// TIA Portal V20 export
FUNCTION_BLOCK "Simulation"   // FB32840, LAD
// stored: MemoryReserve 100, Namespace Unit1.Em8, SetENOAutomatically false
   VAR_INPUT
      simulation { ExternalAccessible := 'False'; ExternalVisible := 'False'; ExternalWritable := 'False'} : Bool;
   END_VAR
   VAR
      instActuator { ExternalAccessible := 'False'; ExternalVisible := 'False'; ExternalWritable := 'False'} : Array[0..9] of "Simulation_Actuator";
      statDigitalSignal { ExternalAccessible := 'False'; ExternalVisible := 'False'; ExternalWritable := 'False'} : Array[0..9] of Bool;
   END_VAR
   VAR_TEMP   // added for the SCL form of the ladder/FBD networks
      _w1 : Bool;
      _w2 : Bool;
      _w3 : Bool;
   END_VAR
BEGIN

REGION Network 1: Digital Signal
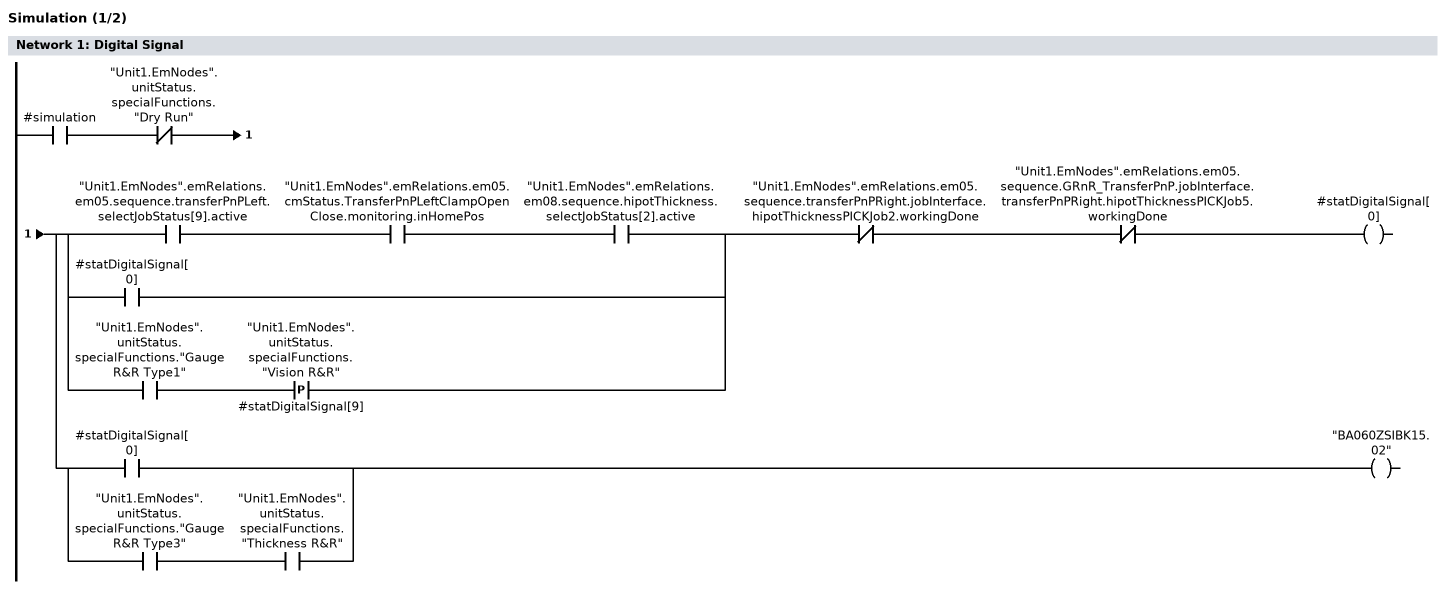
   RUNG wire#powerrail
      Contact( #simulation )
      I_Contact( "Unit1.EmNodes".unitStatus.specialFunctions."Dry Run" )
      wire#w1
      Contact( "Unit1.EmNodes".emRelations.em05.sequence.transferPnPLeft.selectJobStatus[9].active )
      Contact( "Unit1.EmNodes".emRelations.em05.cmStatus.TransferPnPLeftClampOpenClose.monitoring.inHomePos )
      Contact( "Unit1.EmNodes".emRelations.em08.sequence.hipotThickness.selectJobStatus[2].active )
      wire#w2
      I_Contact( "Unit1.EmNodes".emRelations.em05.sequence.transferPnPRight.jobInterface.hipotThicknessPICKJob2.workingDone )
      I_Contact( "Unit1.EmNodes".emRelations.em05.sequence.GRnR_TransferPnP.jobInterface.transferPnPRight.hipotThicknessPICKJob5.workingDone )
      Coil( #statDigitalSignal[0] )
   END_RUNG
   RUNG wire#w1
      Contact( #statDigitalSignal[0] )
   END_RUNG wire#w2
   RUNG wire#w1
      Contact( "Unit1.EmNodes".unitStatus.specialFunctions."Gauge R&R Type1" )
      P_Contact(operand := "Unit1.EmNodes".unitStatus.specialFunctions."Vision R&R", bit := #statDigitalSignal[9])
   END_RUNG wire#w2
   RUNG wire#w1
      Contact( #statDigitalSignal[0] )
      wire#w3
      Coil( "BA060ZSIBK15.02" )
   END_RUNG
   RUNG wire#w1
      Contact( "Unit1.EmNodes".unitStatus.specialFunctions."Gauge R&R Type3" )
      Contact( "Unit1.EmNodes".unitStatus.specialFunctions."Thickness R&R" )
   END_RUNG wire#w3
   // the same network as SCL:
   #_w1 := #simulation AND NOT "Unit1.EmNodes".unitStatus.specialFunctions."Dry Run";
   #_w3 := #_w1 AND #statDigitalSignal[0];
   #_w2 := #_w1 AND "Unit1.EmNodes".unitStatus.specialFunctions."Gauge R&R Type1" AND "Unit1.EmNodes".unitStatus.specialFunctions."Vision R&R" AND NOT #statDigitalSignal[9];   // rising edge of "Unit1.EmNodes".unitStatus.specialFunctions."Vision R&R"
   #statDigitalSignal[9] := "Unit1.EmNodes".unitStatus.specialFunctions."Vision R&R";
   #statDigitalSignal[0] := ((#_w1 AND "Unit1.EmNodes".emRelations.em05.sequence.transferPnPLeft.selectJobStatus[9].active AND "Unit1.EmNodes".emRelations.em05.cmStatus.TransferPnPLeftClampOpenClose.monitoring.inHomePos AND "Unit1.EmNodes".emRelations.em08.sequence.hipotThickness.selectJobStatus[2].active) OR #_w3 OR #_w2) AND NOT "Unit1.EmNodes".emRelations.em05.sequence.transferPnPRight.jobInterface.hipotThicknessPICKJob2.workingDone AND NOT "Unit1.EmNodes".emRelations.em05.sequence.GRnR_TransferPnP.jobInterface.transferPnPRight.hipotThicknessPICKJob5.workingDone;
   "BA060ZSIBK15.02" := #_w1 AND (#statDigitalSignal[0] OR ("Unit1.EmNodes".unitStatus.specialFunctions."Gauge R&R Type3" AND "Unit1.EmNodes".unitStatus.specialFunctions."Thickness R&R"));
END_REGION

REGION Network 2: Two Way Actuator
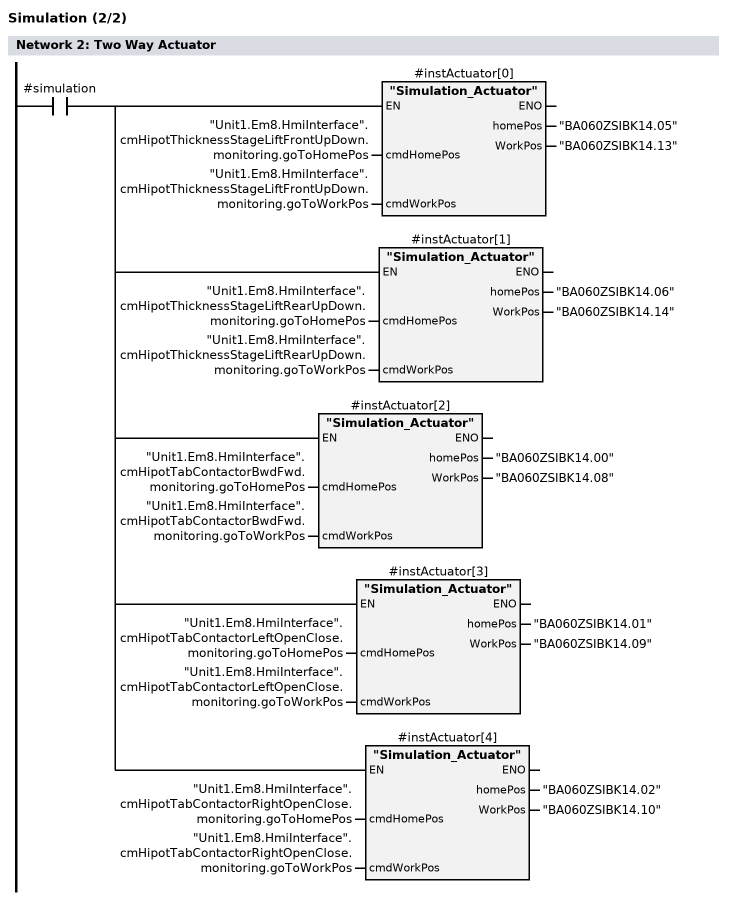
   RUNG wire#powerrail
      Contact( #simulation )
      wire#w1
      #instActuator[0](cmdHomePos := "Unit1.Em8.HmiInterface".cmHipotThicknessStageLiftFrontUpDown.monitoring.goToHomePos, cmdWorkPos := "Unit1.Em8.HmiInterface".cmHipotThicknessStageLiftFrontUpDown.monitoring.goToWorkPos, homePos => "BA060ZSIBK14.05", WorkPos => "BA060ZSIBK14.13")
   END_RUNG
   RUNG wire#w1
      #instActuator[1](cmdHomePos := "Unit1.Em8.HmiInterface".cmHipotThicknessStageLiftRearUpDown.monitoring.goToHomePos, cmdWorkPos := "Unit1.Em8.HmiInterface".cmHipotThicknessStageLiftRearUpDown.monitoring.goToWorkPos, homePos => "BA060ZSIBK14.06", WorkPos => "BA060ZSIBK14.14")
   END_RUNG
   RUNG wire#w1
      #instActuator[2](cmdHomePos := "Unit1.Em8.HmiInterface".cmHipotTabContactorBwdFwd.monitoring.goToHomePos, cmdWorkPos := "Unit1.Em8.HmiInterface".cmHipotTabContactorBwdFwd.monitoring.goToWorkPos, homePos => "BA060ZSIBK14.00", WorkPos => "BA060ZSIBK14.08")
   END_RUNG
   RUNG wire#w1
      #instActuator[3](cmdHomePos := "Unit1.Em8.HmiInterface".cmHipotTabContactorLeftOpenClose.monitoring.goToHomePos, cmdWorkPos := "Unit1.Em8.HmiInterface".cmHipotTabContactorLeftOpenClose.monitoring.goToWorkPos, homePos => "BA060ZSIBK14.01", WorkPos => "BA060ZSIBK14.09")
   END_RUNG
   RUNG wire#w1
      #instActuator[4](cmdHomePos := "Unit1.Em8.HmiInterface".cmHipotTabContactorRightOpenClose.monitoring.goToHomePos, cmdWorkPos := "Unit1.Em8.HmiInterface".cmHipotTabContactorRightOpenClose.monitoring.goToWorkPos, homePos => "BA060ZSIBK14.02", WorkPos => "BA060ZSIBK14.10")
   END_RUNG
   // the same network as SCL:
   IF #simulation THEN
       #instActuator[0](cmdHomePos := "Unit1.Em8.HmiInterface".cmHipotThicknessStageLiftFrontUpDown.monitoring.goToHomePos,   // "Simulation_Actuator"
                        cmdWorkPos := "Unit1.Em8.HmiInterface".cmHipotThicknessStageLiftFrontUpDown.monitoring.goToWorkPos,
                        homePos => "BA060ZSIBK14.05",
                        WorkPos => "BA060ZSIBK14.13");
       #instActuator[1](cmdHomePos := "Unit1.Em8.HmiInterface".cmHipotThicknessStageLiftRearUpDown.monitoring.goToHomePos,   // "Simulation_Actuator"
                        cmdWorkPos := "Unit1.Em8.HmiInterface".cmHipotThicknessStageLiftRearUpDown.monitoring.goToWorkPos,
                        homePos => "BA060ZSIBK14.06",
                        WorkPos => "BA060ZSIBK14.14");
       #instActuator[2](cmdHomePos := "Unit1.Em8.HmiInterface".cmHipotTabContactorBwdFwd.monitoring.goToHomePos,   // "Simulation_Actuator"
                        cmdWorkPos := "Unit1.Em8.HmiInterface".cmHipotTabContactorBwdFwd.monitoring.goToWorkPos,
                        homePos => "BA060ZSIBK14.00",
                        WorkPos => "BA060ZSIBK14.08");
       #instActuator[3](cmdHomePos := "Unit1.Em8.HmiInterface".cmHipotTabContactorLeftOpenClose.monitoring.goToHomePos,   // "Simulation_Actuator"
                        cmdWorkPos := "Unit1.Em8.HmiInterface".cmHipotTabContactorLeftOpenClose.monitoring.goToWorkPos,
                        homePos => "BA060ZSIBK14.01",
                        WorkPos => "BA060ZSIBK14.09");
       #instActuator[4](cmdHomePos := "Unit1.Em8.HmiInterface".cmHipotTabContactorRightOpenClose.monitoring.goToHomePos,   // "Simulation_Actuator"
                        cmdWorkPos := "Unit1.Em8.HmiInterface".cmHipotTabContactorRightOpenClose.monitoring.goToWorkPos,
                        homePos => "BA060ZSIBK14.02",
                        WorkPos => "BA060ZSIBK14.10");
   END_IF;
END_REGION

REGION Network 3 (SCL): homing
   IF #simulation AND "JB_Temp".Test_Homing[8] THEN

       "Unit1.Em8.HmiInterface".cmHipotThicknessStageLiftAllUpDown.commands."commandHomePos" :=
       "Unit1.Em8.HmiInterface".cmThicknessAxisZ.commands.homing := true;

       "JB_Temp".Test_Homing[8] := false;
    //   
   END_IF;

   IF #simulation AND "JB_Temp".Test_Homing[20] THEN


       "Unit1.Em8.HmiInterface".cmHipotThicknessStageLiftAllUpDown.commands."commandHomePos" :=
       "Unit1.Em8.HmiInterface".cmThicknessAxisZ.commands.homing := false;

   END_IF;
END_REGION
END_FUNCTION_BLOCK
